	(* payload rear string *)
	str	:= ',"payload_rear":[';
	FOR i:=1 TO Get_Data.Data_Length BY 1 DO
		CONCAT2(ADR(str), ADR(Get_Data.Payload_Rear[i]), ADR(str), SIZEOF(str)); 
		
		IF i <> Get_Data.Data_Length THEN
			CONCAT2(ADR(str), ADR(comma), ADR(str), SIZEOF(str));
		ELSE
			CONCAT2(ADR(str), ADR(arrayEnd2), ADR(str), SIZEOF(str));
		END_IF
		
	END_FOR
	
	CONCAT2(ADR(sPayloadPub), ADR(str), ADR(sPayloadPub), SIZEOF(sPayloadPub));
	
	(* overload lead string *)
	str	:= ',"overload_lead":[';
	FOR i:=1 TO Get_Data.Data_Length BY 1 DO
		CONCAT2(ADR(str), ADR(Get_Data.Overload_Lead[i]), ADR(str), SIZEOF(str)); 
		
		IF i <> Get_Data.Data_Length THEN
			CONCAT2(ADR(str), ADR(comma), ADR(str), SIZEOF(str));
		ELSE
			CONCAT2(ADR(str), ADR(arrayEnd2), ADR(str), SIZEOF(str));
		END_IF
		
	END_FOR
	
	CONCAT2(ADR(sPayloadPub), ADR(str), ADR(sPayloadPub), SIZEOF(sPayloadPub));
	
	(* overload rear string *)
	str	:= ',"overload_rear":[';
	FOR i:=1 TO Get_Data.Data_Length BY 1 DO
		CONCAT2(ADR(str), ADR(Get_Data.Overload_Rear[i]), ADR(str), SIZEOF(str)); 
		
		IF i <> Get_Data.Data_Length THEN
			CONCAT2(ADR(str), ADR(comma), ADR(str), SIZEOF(str));
		ELSE
			CONCAT2(ADR(str), ADR(arrayEnd2), ADR(str), SIZEOF(str));
		END_IF
		
	END_FOR
	
	CONCAT2(ADR(sPayloadPub), ADR(str), ADR(sPayloadPub), SIZEOF(sPayloadPub));
	
	(* pressure lead string *)
	str	:= ',"pressure_lead":[';
	FOR i:=1 TO Get_Data.Data_Length BY 1 DO
		CONCAT2(ADR(str), ADR(Get_Data.Pressure_Lead[i]), ADR(str), SIZEOF(str)); 
		
		IF i <> Get_Data.Data_Length THEN
			CONCAT2(ADR(str), ADR(comma), ADR(str), SIZEOF(str));
		ELSE
			CONCAT2(ADR(str), ADR(arrayEnd2), ADR(str), SIZEOF(str));
		END_IF
		
	END_FOR
	
	CONCAT2(ADR(sPayloadPub), ADR(str), ADR(sPayloadPub), SIZEOF(sPayloadPub));

	(* pressure rear string *)
	str	:= ',"pressure_rear":[';
	FOR i:=1 TO Get_Data.Data_Length BY 1 DO
		CONCAT2(ADR(str), ADR(Get_Data.Pressure_Rear[i]), ADR(str), SIZEOF(str)); 
		
		IF i <> Get_Data.Data_Length THEN
			CONCAT2(ADR(str), ADR(comma), ADR(str), SIZEOF(str));
		ELSE
			CONCAT2(ADR(str), ADR(arrayEnd2), ADR(str), SIZEOF(str));
		END_IF
		
	END_FOR
	
	CONCAT2(ADR(sPayloadPub), ADR(str), ADR(sPayloadPub), SIZEOF(sPayloadPub));
	
	(* overpressure lead string *)
	str	:= ',"overpressure_lead":[';
	FOR i:=1 TO Get_Data.Data_Length BY 1 DO
		CONCAT2(ADR(str), ADR(Get_Data.Overpressure_Lead[i]), ADR(str), SIZEOF(str)); 
		
		IF i <> Get_Data.Data_Length THEN
			CONCAT2(ADR(str), ADR(comma), ADR(str), SIZEOF(str));
		ELSE
			CONCAT2(ADR(str), ADR(arrayEnd2), ADR(str), SIZEOF(str));
		END_IF
		
	END_FOR
	
	CONCAT2(ADR(sPayloadPub), ADR(str), ADR(sPayloadPub), SIZEOF(sPayloadPub));
	
	(* overpressure rear string *)
	str	:= ',"overpressure_rear":[';
	FOR i:=1 TO Get_Data.Data_Length BY 1 DO
		CONCAT2(ADR(str), ADR(Get_Data.Overpressure_Rear[i]), ADR(str), SIZEOF(str)); 
		
		IF i <> Get_Data.Data_Length THEN
			CONCAT2(ADR(str), ADR(comma), ADR(str), SIZEOF(str));
		ELSE
			CONCAT2(ADR(str), ADR(arrayEnd2), ADR(str), SIZEOF(str));
		END_IF
		
	END_FOR
	
	CONCAT2(ADR(sPayloadPub), ADR(str), ADR(sPayloadPub), SIZEOF(sPayloadPub));
	
	(* event code string *)
	str	:= ',"event_code":[';
	FOR i:=1 TO Get_Data.Data_Length BY 1 DO
		CONCAT2(ADR(str), ADR(Get_Data.EventCode[i]), ADR(str), SIZEOF(str)); 
		
		IF i <> Get_Data.Data_Length THEN
			CONCAT2(ADR(str), ADR(comma), ADR(str), SIZEOF(str));
		ELSE
			CONCAT2(ADR(str), ADR(arrayEnd2), ADR(str), SIZEOF(str));
		END_IF
		
	END_FOR
	
	CONCAT2(ADR(sPayloadPub), ADR(str), ADR(sPayloadPub), SIZEOF(sPayloadPub));
	
	CONCAT2(ADR(sPayloadPub), ADR(msgEnd), ADR(sPayloadPub), SIZEOF(sPayloadPub)); //message ending
	
	(* publish message to subscribed topic *)
	IF Publish := fbMqttClient.Publish(sTopic:= sTopicPub, pPayload:= ADR(sPayloadPub), nPayloadSize:= LEN2(ADR(sPayloadPub)), eQoS:= TcIotMqttQos.AtMostOnceDelivery, bRetain:= FALSE, bQueue:= FALSE) THEN
		IF fbMqttClient.bError THEN
			// add your error logging here			
			hrErrorOccurred := fbMqttClient.hrErrorCode;
		ELSE
			Published 	:= TRUE;
		END_IF
		
	END_IF
	
END_IF

END_PROGRAM

// ---- POUs/Save_Data.TcPOU
PROGRAM Save_Data
VAR
	fbSqlDatabase	: FB_SQLDatabaseEvt(sNetID := '', tTimeout := T#1000S);
	fbSqlCommand	: FB_SQLCommandEvt(sNetID := '', tTimeout := T#1000S);
	fbSqlResult		: FB_SQLResultEvt(sNetID:='', tTimeout   := T#1000S); 
	sCmd			: STRING(100000);
	sCmd2			: STRING(10000);
	nState			: INT;
	
	Done			: BOOL;
	i				: ULINT;
	Vacuumed		: BOOL := FALSE;
	
	aReadStruct		: ST_SelectStructData;
	Oldest_data		: DWORD;
	Today			: DWORD;
	
	Deleted			: BOOL;
	Pragma_Done		: BOOL;
END_VAR

(* connect to localdb *)
IF NOT fbSqlDatabase.bConnected THEN
	fbSqlDatabase.Connect(3);
ELSE

	CASE nState OF
				
		0:
			Done := FALSE;
			IF fbSqlDatabase.CreateCmd(ADR(fbSqlCommand)) THEN
				IF fbSqlDatabase.bError THEN
					nState := 255; 
				ELSE
					IF NOT Deleted THEN
						nState := nState+1;
					ELSE
						nState := 6; //skip to save data
					END_IF
				END_IF
			END_IF
			
		1:	(* execute pragmas *)
			IF NOT Pragma_Done THEN
				sCmd	:= 'PRAGMA journal_mode = WAL; PRAGMA synchronous = NORMAL; PRAGMA temp_store = MEMORY; PRAGMA mmap_size = 30000000000; PRAGMA page_size = 32768; PRAGMA locking_mode = EXCLUSIVE;';
			
				IF fbSQLCommand.Execute(ADR(sCmd), SIZEOF(sCmd)) THEN
					IF fbSQLCommand.bError THEN
						nState := 255; 
					ELSE
						nState 		:= nState+1; 
						Pragma_Done := TRUE;
					END_IF
				END_IF
			
			ELSE
				nState 		:= nState+1;
			END_IF
			
		2:
			(* select oldest data from buffer_imu *)
			sCmd	:= 'SELECT * FROM `data` ORDER BY datetime ASC LIMIT 1';
			
			IF fbSQLCommand.ExecuteDataReturn(ADR(sCmd), SIZEOF(sCmd), ADR(fbSqlResult)) THEN
				IF fbSQLCommand.bError THEN
					nState := 255; 
				ELSE
					nState := nState+1; 
				END_IF
			END_IF
			
		3:
			IF fbSqlResult.Read(0, 1, ADR(aReadStruct), SIZEOF(aReadStruct), TRUE, TRUE) THEN
				IF fbSqlResult.bError THEN
					nState := 255; 
				ELSE
					nState := nState+1; 
				END_IF
			END_IF
			
		4:
			IF fbSqlResult.Release() THEN
				IF fbSqlResult.bError THEN
					nState := 255;
				ELSE
					nState := nState+1;
				END_IF
			END_IF
			
		5:	
			//oldest data < today - 3 months?
			aReadStruct.datetime 	:= REPLACE(aReadStruct.datetime, '-', 1, 11);
			Oldest_data				:= DT_TO_DWORD(SYSTEMTIME_TO_DT(STRING_TO_SYSTEMTIME(aReadStruct.datetime)));
			Today					:= DT_TO_DWORD(SYSTEMTIME_TO_DT(Background_Time.fbTime.systemTime));
			
			IF Oldest_data < (Today - 7776000) THEN
				sCmd	:= 'DELETE FROM data WHERE datetime < datetime($'now$', $'-3 month$');';
		
				IF fbSQLCommand.Execute(ADR(sCmd), SIZEOF(sCmd)) THEN
					IF fbSQLCommand.bError THEN
						nState := 255; 
					ELSE
						nState 	:= nState+1;
						Deleted	:= TRUE;
					END_IF
					
				END_IF
			ELSE
				nState 	:= nState+1;
				Deleted	:= TRUE;
			END_IF
			
		6:	
			(* build query *)	
			sCmd	:= 'INSERT INTO data (datetime,trailer_id_lead,trailer_id_rear,latitude,longitude,speed,overspeed,payload_lead,payload_rear,overload_lead,overload_rear,pressure_lead,pressure_rear,overpressure_lead,overpressure_rear,event_code) VALUES ';
			
			FOR i := 1 TO Get_Data.Data_Length BY 1 DO
					sCmd2:= CONCAT('($'', Get_Data.TimeStr[i]);
					sCmd2:= CONCAT(sCmd2, '$',');
					sCmd2:= CONCAT(sCmd2, Get_Data.Trailer_ID_Lead[i]);
					sCmd2:= CONCAT(sCmd2, ',');
					sCmd2:= CONCAT(sCmd2, Get_Data.Trailer_ID_Rear[i]);
					sCmd2:= CONCAT(sCmd2, ',');
					sCmd2:= CONCAT(sCmd2, Get_Data.Lat[i]);
					sCmd2:= CONCAT(sCmd2, ',');
					sCmd2:= CONCAT(sCmd2, Get_Data.Lon[i]);
					sCmd2:= CONCAT(sCmd2, ',');
					sCmd2:= CONCAT(sCmd2, Get_Data.Speed[i]);
					sCmd2:= CONCAT(sCmd2, ',');
					sCmd2:= CONCAT(sCmd2, Get_Data.Overspeed[i]);
					sCmd2:= CONCAT(sCmd2, ',');
					sCmd2:= CONCAT(sCmd2, Get_Data.Payload_Lead[i]);
					sCmd2:= CONCAT(sCmd2, ',');
					sCmd2:= CONCAT(sCmd2, Get_Data.Payload_Rear[i]);
					sCmd2:= CONCAT(sCmd2, ',');
					sCmd2:= CONCAT(sCmd2, Get_Data.Overload_Lead[i]);
					sCmd2:= CONCAT(sCmd2, ',');
					sCmd2:= CONCAT(sCmd2, Get_Data.Overload_Rear[i]);
					sCmd2:= CONCAT(sCmd2, ',');
					sCmd2:= CONCAT(sCmd2, Get_Data.Pressure_Lead[i]); 
					sCmd2:= CONCAT(sCmd2, ',');
					sCmd2:= CONCAT(sCmd2, Get_Data.Pressure_Rear[i]); 
					sCmd2:= CONCAT(sCmd2, ',');
					sCmd2:= CONCAT(sCmd2, Get_Data.Overpressure_Lead[i]); 
					sCmd2:= CONCAT(sCmd2, ',');
					sCmd2:= CONCAT(sCmd2, Get_Data.Overpressure_Rear[i]); 
					sCmd2:= CONCAT(sCmd2, ',');
					sCmd2:= CONCAT(sCmd2, Get_Data.EventCode[i]);
					
					IF i = Get_Data.Data_Length THEN
						sCmd2:= CONCAT(sCmd2, ')');
					ELSE	
						sCmd2:= CONCAT(sCmd2, '),');
					END_IF
					
					CONCAT2(ADR(sCmd), ADR(sCmd2), ADR(sCmd), SIZEOF(sCmd));
				END_FOR
			
			IF fbSQLCommand.Execute(ADR(sCmd), SIZEOF(sCmd)) THEN
				IF fbSQLCommand.bError THEN
					nState := 255; 
				ELSE
					nState := nState+1; 
					
					
				END_IF
			END_IF
		
		7: 
			Done	:= TRUE;
			nState	:= 0;
				
		255:
			nState := 0;
	
	END_CASE
	
	(*
	CASE nState OF
				
		0:
			Done := FALSE;
			IF fbSqlDatabase.CreateCmd(ADR(fbSqlCommand)) THEN
				IF fbSqlDatabase.bError THEN
					nState := 255; 
				ELSE
					nState := nState+1; 
				END_IF
			END_IF
			
		1:	
			(* build query *)	
			sCmd	:= 'DELETE FROM data WHERE datetime < datetime($'now$', $'-3 month$');';
			
			IF fbSQLCommand.Execute(ADR(sCmd), SIZEOF(sCmd)) THEN
				IF fbSQLCommand.bError THEN
					nState := 255; 
				ELSE
					nState := nState+1; 
					
					
				END_IF
			END_IF
			
		2:	
			(* build query *)	
			sCmd	:= 'INSERT INTO data (datetime,trailer_id_lead,trailer_id_rear,latitude,longitude,speed,overspeed,payload_lead,payload_rear,overload_lead,overload_rear,pressure_lead,pressure_rear,overpressure_lead,overpressure_rear,event_code) VALUES ';
			
			FOR i := 1 TO Get_Data.Data_Length BY 1 DO
					sCmd2:= CONCAT('($'', Get_Data.TimeStr[i]);
					sCmd2:= CONCAT(sCmd2, '$',');
					sCmd2:= CONCAT(sCmd2, Get_Data.Trailer_ID_Lead[i]);
					sCmd2:= CONCAT(sCmd2, ',');
					sCmd2:= CONCAT(sCmd2, Get_Data.Trailer_ID_Rear[i]);
					sCmd2:= CONCAT(sCmd2, ',');
					sCmd2:= CONCAT(sCmd2, Get_Data.Lat[i]);
					sCmd2:= CONCAT(sCmd2, ',');
					sCmd2:= CONCAT(sCmd2, Get_Data.Lon[i]);
					sCmd2:= CONCAT(sCmd2, ',');
					sCmd2:= CONCAT(sCmd2, Get_Data.Speed[i]);
					sCmd2:= CONCAT(sCmd2, ',');
					sCmd2:= CONCAT(sCmd2, Get_Data.Overspeed[i]);
					sCmd2:= CONCAT(sCmd2, ',');
					sCmd2:= CONCAT(sCmd2, Get_Data.Payload_Lead[i]);
					sCmd2:= CONCAT(sCmd2, ',');
					sCmd2:= CONCAT(sCmd2, Get_Data.Payload_Rear[i]);
					sCmd2:= CONCAT(sCmd2, ',');
					sCmd2:= CONCAT(sCmd2, Get_Data.Overload_Lead[i]);
					sCmd2:= CONCAT(sCmd2, ',');
					sCmd2:= CONCAT(sCmd2, Get_Data.Overload_Rear[i]);
					sCmd2:= CONCAT(sCmd2, ',');
					sCmd2:= CONCAT(sCmd2, Get_Data.Pressure_Lead[i]); 
					sCmd2:= CONCAT(sCmd2, ',');
					sCmd2:= CONCAT(sCmd2, Get_Data.Pressure_Rear[i]); 
					sCmd2:= CONCAT(sCmd2, ',');
					sCmd2:= CONCAT(sCmd2, Get_Data.Overpressure_Lead[i]); 
					sCmd2:= CONCAT(sCmd2, ',');
					sCmd2:= CONCAT(sCmd2, Get_Data.Overpressure_Rear[i]); 
					sCmd2:= CONCAT(sCmd2, ',');
					sCmd2:= CONCAT(sCmd2, Get_Data.EventCode[i]);
					
					IF i = Get_Data.Data_Length THEN
						sCmd2:= CONCAT(sCmd2, ')');
					ELSE	
						sCmd2:= CONCAT(sCmd2, '),');
					END_IF
					
					CONCAT2(ADR(sCmd), ADR(sCmd2), ADR(sCmd), SIZEOF(sCmd));
				END_FOR
			
			IF fbSQLCommand.Execute(ADR(sCmd), SIZEOF(sCmd)) THEN
				IF fbSQLCommand.bError THEN
					nState := 255; 
				ELSE
					nState := nState+1; 
					
					
				END_IF
			END_IF
				
		3: 
			Done	:= TRUE;
			nState	:= 0;
				
		255:
			nState := 0;
	
	END_CASE
	*)
	
END_IF

END_PROGRAM

// ---- POUs/Main_Vacuum.TcPOU
PROGRAM Main_Vacuum
VAR
END_VAR

IF NOT Vacuum_Buffer_Data.Vacuumed THEN
	Vacuum_Buffer_Data();
END_IF

IF NOT Vacuum_Buffer_IMU.Vacuumed THEN
	Vacuum_Buffer_IMU();
END_IF

IF NOT Vacuum_Buffer_IMU_2.Vacuumed THEN
	Vacuum_Buffer_IMU_2();
END_IF

IF NOT Vacuum_Data.Vacuumed THEN
	Vacuum_Data();
END_IF

IF NOT Vacuum_IMU.Vacuumed THEN
	Vacuum_IMU();
END_IF

END_PROGRAM

// ---- POUs/Vacuum_Data.TcPOU
PROGRAM Vacuum_Data
VAR
	fbSqlDatabase	: FB_SQLDatabaseEvt(sNetID := '', tTimeout := T#1000S);
	fbSqlCommand	: FB_SQLCommandEvt(sNetID := '', tTimeout := T#1000S);
	fbSqlResult		: FB_SQLResultEvt(sNetID :='', tTimeout   := T#1000S); 
	nState			: INT;
	sCmd			: STRING(500000);
	Vacuumed		: BOOL;
END_VAR

CASE nState OF
				
		0:
			(* connect to buffer_imu *)		
			IF fbSqlDatabase.Connect(3) THEN
				IF fbSqlDatabase.bError THEN
					nState := 255; 
				ELSE
					IF fbSqlDatabase.bConnected THEN
						nState := nState+1;
					END_IF 
				END_IF
			END_IF
			
		1:
			IF fbSqlDatabase.CreateCmd(ADR(fbSqlCommand)) THEN
				IF fbSqlDatabase.bError THEN
					nState := 255; 
				ELSE
					nState := nState+1; 
				END_IF
			END_IF
			
		2:	(* execute pragmas *)
			sCmd	:= 'PRAGMA journal_mode = WAL; PRAGMA synchronous = NORMAL; PRAGMA temp_store = MEMORY; PRAGMA mmap_size = 30000000000; PRAGMA page_size = 32768; PRAGMA locking_mode = EXCLUSIVE;';
			
			IF fbSQLCommand.Execute(ADR(sCmd), SIZEOF(sCmd)) THEN
				IF fbSQLCommand.bError THEN
					nState := 255; 
				ELSE
					nState := nState+1; 
				END_IF
			END_IF
		
		3:	
			IF NOT Vacuumed THEN
				(* build query *)	
				sCmd	:= 'VACUUM';
				
				IF fbSQLCommand.Execute(ADR(sCmd), SIZEOF(sCmd)) THEN
					IF fbSQLCommand.bError THEN
						nState := 255; 
					ELSE
						nState 		:= nState+1; 
					END_IF
				END_IF
				
			ELSE 
				nState := nState+1;
			END_IF
			
		4:	(* execute pragma optimize *)
			sCmd	:= 'PRAGMA optimize;';
			
			IF fbSQLCommand.Execute(ADR(sCmd), SIZEOF(sCmd)) THEN
				IF fbSQLCommand.bError THEN
					nState := 255; 
				ELSE
					nState := nState+1; 
				END_IF
			END_IF
		
		5:
			IF fbSqlDatabase.Disconnect() THEN
				IF fbSqlDatabase.bError THEN
					nState := 255;
				ELSE
					nState 		:= nState+1;
					Vacuumed 	:= TRUE;
				END_IF
			END_IF
			
		255:
			nState := 0;
			
END_CASE

END_PROGRAM
